{attribute 'enable_dynamic_creation'}
TYPE ST_ActionStatus :
STRUCT
	nActionId	: UINT;
	eAction		: E_Action;
	nObjectId	: UINT;
	eStatus		: E_ActionStatus;
	nChannel	: USINT;
	eOldStatus	: E_ActionStatus;
END_STRUCT
END_TYPE

(* stored: Version 1.1.0.1, ProductVersion 3.1.4022.10
   DUT ST_ActionStatus: Id {3e565aba-943f-4d6a-bbb5-bcc8871753c6} *)
